FUNCTION_BLOCK FB_Snake
VAR_IN_OUT
	//first item is head
	aStSnakeBody	: ARRAY[1..GVL_Constants.SNAKE_LENGTH] OF ST_SnakePart;
	iSnakeLength 	: INT;
END_VAR
VAR_OUTPUT
END_VAR
VAR
	
END_VAR

METHOD M_Die : BOOL
VAR_INPUT
END_VAR

VAR
	iPartIndex: INT;
END_VAR
{warning disable C0371}
IF NOT __ISVALIDREF(aStSnakeBody) AND NOT __ISVALIDREF(iSnakeLength) THEN
     RETURN;
END_IF

M_Die := FALSE;
IF aStSnakeBody[1].stBodyCoordinate.iColumnCoordinate > 9 OR aStSnakeBody[1].stBodyCoordinate.iColumnCoordinate < 0 OR
	aStSnakeBody[1].stBodyCoordinate.iRowCoordinate < 0 OR aStSnakeBody[1].stBodyCoordinate.iRowCoordinate > 9 THEN
	M_Die := TRUE;
END_IF

IF iSnakeLength >= 4 THEN
	FOR iPartIndex := iSnakeLength TO 2 BY -1 DO
		IF aStSnakeBody[1].stBodyCoordinate.iColumnCoordinate = aStSnakeBody[iPartIndex].stBodyCoordinate.iColumnCoordinate AND
			aStSnakeBody[1].stBodyCoordinate.iRowCoordinate = aStSnakeBody[iPartIndex].stBodyCoordinate.iRowCoordinate THEN
			M_Die := TRUE;
		END_IF
	END_FOR
END_IF

{warning restore C0371}
END_METHOD

//if head cordinate and food cordinate match then snake has eaten the food and got larger
METHOD PUBLIC M_Eat : BOOL
VAR_INPUT
	stFood		: ST_Food;
END_VAR
VAR
	bHasEaten	: BOOL;
END_VAR
{warning disable C0371}
IF NOT __ISVALIDREF(aStSnakeBody) AND NOT __ISVALIDREF(iSnakeLength) THEN
     RETURN;
END_IF

IF aStSnakeBody[1].stBodyCoordinate.iColumnCoordinate = stFood.stFoodCoordinate.iColumnCoordinate AND
	aStSnakeBody[1].stBodyCoordinate.iRowCoordinate = stFood.stFoodCoordinate.iRowCoordinate THEN	
	bHasEaten := TRUE;
ELSE
	bHasEaten := FALSE;
END_IF

IF bHasEaten AND iSnakeLength <= GVL_Constants.SNAKE_LENGTH THEN
	iSnakeLength := iSnakeLength + 1;
END_IF

M_Eat := bHasEaten;
{warning restore C0371}
END_METHOD

METHOD PUBLIC M_Move : BOOL
VAR_INPUT
	iHeadDirection : INT;
END_VAR

VAR
	bMoved			: BOOL;
	iPartIndex		: INT;
END_VAR
{warning disable C0371}
M_Move := FALSE;
IF NOT __ISVALIDREF(THIS^.aStSnakeBody) AND NOT __ISVALIDREF(iSnakeLength) THEN
     RETURN;
END_IF

FOR iPartIndex := iSnakeLength+1 TO 2 BY -1 DO
	aStSnakeBody[iPartIndex].stBodyCoordinate := aStSnakeBody[iPartIndex - 1].stBodyCoordinate;
END_FOR

IF iHeadDirection = 1 THEN	
	bMoved	:= TRUE;
	aStSnakeBody[1].stBodyCoordinate.iColumnCoordinate	:= aStSnakeBody[1].stBodyCoordinate.iColumnCoordinate - 1;
ELSIF iHeadDirection = 4  THEN
	bMoved	:= TRUE;
	aStSnakeBody[1].stBodyCoordinate.iColumnCoordinate := aStSnakeBody[1].stBodyCoordinate.iColumnCoordinate + 1;
ELSIF iHeadDirection = 3  THEN
	bMoved	:= TRUE;
	aStSnakeBody[1].stBodyCoordinate.iRowCoordinate	:=  aStSnakeBody[1].stBodyCoordinate.iRowCoordinate + 1;
ELSIF iHeadDirection = 2 THEN
	bMoved	:= TRUE;
	aStSnakeBody[1].stBodyCoordinate.iRowCoordinate	:= aStSnakeBody[1].stBodyCoordinate.iRowCoordinate - 1;
END_IF
M_Move := bMoved;
{warning restore C0371}
END_METHOD

END_FUNCTION_BLOCK

(* stored: Version 1.1.0.1, ProductVersion 3.1.4024.4
   POU FB_Snake: Id {3c39ea80-2fff-43f9-91a7-1fc592c0813c}, SpecialFunc None
   Method M_Die: Id {620e688c-30e0-4e36-8e15-483fe31cd1f5}
   Method M_Eat: Id {7391ae2d-e7c4-48a5-8d76-0e7f4e7388f4}
   Method M_Move: Id {e591df98-d7b0-47dc-8b98-5284189e1612} *)
